// TIA Portal V19 export
DATA_BLOCK "1200 Comm_DB"   // DB2
// stored: InstanceOfName 1200 Comm, InstanceOfType FB
"1200 Comm"
BEGIN
END_DATA_BLOCK
